PROGRAM MAIN
VAR
	TestBitsArr		: ARRAY [0..72] OF BOOL;
	bCalc: BOOL;
	CountedTrueBits		: UINT;
	MyBitsArrSize: UINT;
END_VAR


IF bCalc THEN
	MyBitsArrSize	:= SIZEOF(TestBitsArr);
	CountedTrueBits:= F_TrueBitsCounter(pArray:= ADR(TestBitsArr),arrBitSize:= MyBitsArrSize);
	bCalc			:= FALSE;
END_IF

END_PROGRAM

(* stored: Version 1.1.0.1, ProductVersion 3.1.4024.12
   POU MAIN: Id {6a4d60f6-2cbe-4291-af71-7fb03a1327c1}, SpecialFunc None *)
